// TIA Portal project "PLCwirelessCtrl" (V17)

(* hardware
DEVICE "ET 200SP-Station_1"  ET 200SP-Station
   slot 0: "Baugruppenträger_0"  Rack  6ES5 710-8MAx1
   slot 1: "PLC_1"  CPU 1510SP-1 PN  6ES7 510-1DJ01-0AB0  V2.5
      slot 32768: "PROFINET-Schnittstelle_1"  X1
         slot 32771: "Port_3"  X1 P3
   slot 2: "Servermodul_1"  Server module  6ES7 193-6PA00-0AA0  V1.1
      slot 1: "Servermodul_1"  Server module
   slot 127: "BA 2xRJ45"  BA 2xRJ45  6ES7 193-6AR00-0AA0  V0.0
      slot 32769: "Port_1"  X1 P1  6ES7 193-6AR00-0AA0
      slot 32770: "Port_2"  X1 P2  6ES7 193-6AR00-0AA0
*)

// ===== PLC "PLC_1"  CPU 1510SP-1 PN =====

VAR_GLOBAL   // PLC tag table "Standard-Variablentabelle"
   "Tag_1" AT %M10.1 : Bool;
END_VAR

TYPE "stateBool"
   STRUCT
      "name" : String;
      value : Bool := false;
      alarm : Bool;
      visible : Bool;
      "type" : String := 'bool';
      si : String;
   END_STRUCT;
END_TYPE

TYPE "stateInt"
   STRUCT
      "name" : String;
      value : Int := 52;
      alarm : Bool;
      visible : Bool;
      "type" : String;
      si : String;
   END_STRUCT;
END_TYPE

TYPE "stateReal"
   STRUCT
      "name" : String;
      value : Real := 456.43;
      alarm : Bool;
      visible : Bool;
      "type" : String;
      si : String := '[mbar]';
   END_STRUCT;
END_TYPE

TYPE "paraInt"
   STRUCT
      "name" : String;
      value : Int := 0;
      input : Int;
      locked : Bool := false;
      min : Int := 0;
      max : Int := 9999;
      visible : Bool := true;
      newVal : Bool;
      "type" : String := 'int';
      add : String;
      si : String;
      new : Bool;
   END_STRUCT;
END_TYPE

TYPE "paraBool"
   STRUCT
      "name" : String;
      value : Bool := 0;
      input : Bool;
      locked : Bool := false;
      min : Int := 0;
      max : Int := 1;
      visible : Bool := true;
      newVal : Bool;
      "type" : String := 'bool';
      add : String;
      si : String;
      new : Bool;
   END_STRUCT;
END_TYPE

TYPE "paraReal"
   STRUCT
      "name" : String;
      value : Real := 0.0;
      input : Real;
      locked : Bool := false;
      min : Real := 0.0;
      max : Real := 9999.99;
      visible : Bool := true;
      newVal : Bool;
      "type" : String := 'real';
      add : String;
      si : String;
      new : Bool;
   END_STRUCT;
END_TYPE

TYPE "function"
   STRUCT
      "name" : String;
      active : Bool;
      locked : Bool;
      visible : Bool;
      fault : Bool;
      button : Bool;
      add : Bool;
   END_STRUCT;
END_TYPE

DATA_BLOCK "handleWebserverDat_DB"   // DB1
{ S7_Optimized_Access := 'TRUE' }
VERSION : 0.1
// stored: InstanceOfName handleWebserverDat
"handleWebserverDat"
BEGIN
END_DATA_BLOCK

DATA_BLOCK "webserverData"   // DB3
{ S7_Optimized_Access := 'TRUE' }
VERSION : 0.1
   VAR
      fct00 : "function";
      fct01 : "function";
      fct02 : "function";
      fct03 : "function";
      fct04 : "function";
      fct05 : "function";
      fct06 : "function";
      fct07 : "function";
      fct08 : "function";
      fct09 : "function";
      par00 : "paraInt";
      par01 : "paraBool";
      par02 : "paraReal";
      par03 : "paraInt";
      par04 : "paraInt";
      par05 : "paraInt";
      par06 : "paraInt";
      par07 : "paraInt";
      par08 : "paraInt";
      par09 : "paraInt";
      sta01 : "stateBool";
      sta00 : "stateReal";
      sta02 : "stateBool";
      sta03 : "stateBool";
      sta04 : "stateBool";
      sta05 : "stateBool";
      sta06 : "stateBool";
      sta07 : "stateInt";
      sta08 : "stateBool";
      sta09 : "stateBool";
      alr : Array[0..19] of String;
   END_VAR
BEGIN
   par00."name" := 'Setpoint 1';
   par00."type" := 'int';
   sta01.visible := TRUE;
   sta00."name" := 'Pressure Value';
   sta00.visible := TRUE;
   sta02.value := TRUE;
   sta02.visible := TRUE;
   sta02."type" := 'bool';
   sta07."name" := 'Integer Number';
   sta07.value := 523;
   sta07.si := 'Dig';
   sta01.si := 'Seconds';
   sta01."name" := 'Status of Function';
   par00.min := 0;
   par00.max := 100;
   par00.si := 'cycles';
   par01."name" := 'Manual Mode';
   par02."name" := 'Level';
   par02.si := 'm';
   par02.min := 0.0;
   par02.max := 2000.0;
   par02.locked := TRUE;
   par03."name" := 'Locked Parameter';
   par03.min := 60;
   par03.max := 70;
   par03.locked := TRUE;
   par03.si := 'rpm';
   fct00.visible := TRUE;
   fct01.active := TRUE;
   fct02.locked := TRUE;
   fct03.active := TRUE;
   fct03.locked := TRUE;
   fct03.visible := TRUE;
   fct02.visible := TRUE;
   fct01.visible := TRUE;
   fct04.visible := TRUE;
   fct04.fault := TRUE;
   fct00."name" := 'Function 1';
   fct01."name" := 'Function 2';
   fct02."name" := 'Activate Pump';
   fct03."name" := 'Start Purge';
   fct04."name" := 'Function in Error';
   fct05."name" := 'Reset';
   fct06."name" := 'Do Something';
   fct07."name" := 'Function 8';
   fct08."name" := 'Not Visible';
   fct09."name" := 'Function 10';
   fct09.visible := TRUE;
   fct06.visible := TRUE;
   fct07.visible := TRUE;
   fct05.visible := TRUE;
   sta01."type" := 'bool';
   sta06."name" := 'Distance';
   sta06."type" := 'bool';
   sta06.si := 'm';
   sta00.si := '(mbar)';
   fct00.active := FALSE;
   fct00.locked := FALSE;
   fct00.fault := FALSE;
   fct00.button := FALSE;
   fct00.add := FALSE;
   fct01.locked := FALSE;
   fct01.fault := FALSE;
   fct01.button := FALSE;
   fct01.add := FALSE;
   fct02.active := FALSE;
   fct02.fault := FALSE;
   fct02.button := FALSE;
   fct02.add := FALSE;
   fct03.fault := FALSE;
   fct03.button := FALSE;
   fct03.add := FALSE;
   fct04.active := FALSE;
   fct04.locked := FALSE;
   fct04.button := FALSE;
   fct04.add := FALSE;
   fct05.active := FALSE;
   fct05.locked := FALSE;
   fct05.fault := FALSE;
   fct05.button := FALSE;
   fct05.add := FALSE;
   fct06.active := FALSE;
   fct06.locked := FALSE;
   fct06.fault := FALSE;
   fct06.button := FALSE;
   fct06.add := FALSE;
   fct07.active := FALSE;
   fct07.locked := FALSE;
   fct07.fault := FALSE;
   fct07.button := FALSE;
   fct07.add := FALSE;
   fct08.active := FALSE;
   fct08.locked := FALSE;
   fct08.visible := FALSE;
   fct08.fault := FALSE;
   fct08.button := FALSE;
   fct08.add := FALSE;
   fct09.active := FALSE;
   fct09.locked := FALSE;
   fct09.fault := FALSE;
   fct09.button := FALSE;
   fct09.add := FALSE;
   par00.value := 0;
   par00.input := 0;
   par00.locked := FALSE;
   par00.visible := TRUE;
   par00.newVal := FALSE;
   par00.add := '';
   par00.new := FALSE;
   par01.value := FALSE;
   par01.input := FALSE;
   par01.locked := FALSE;
   par01.min := 0;
   par01.max := 1;
   par01.visible := TRUE;
   par01.newVal := FALSE;
   par01."type" := 'bool';
   par01.add := '';
   par01.si := '';
   par01.new := FALSE;
   par02.value := 0.0;
   par02.input := 0.0;
   par02.visible := TRUE;
   par02.newVal := FALSE;
   par02."type" := 'real';
   par02.add := '';
   par02.new := FALSE;
   par03.value := 0;
   par03.input := 0;
   par03.visible := TRUE;
   par03.newVal := FALSE;
   par03."type" := 'int';
   par03.add := '';
   par03.new := FALSE;
   par04."name" := '';
   par04.value := 0;
   par04.input := 0;
   par04.locked := FALSE;
   par04.min := 0;
   par04.max := 9999;
   par04.visible := FALSE;
   par04.newVal := FALSE;
   par04."type" := 'int';
   par04.add := '';
   par04.si := '';
   par04.new := FALSE;
   par05."name" := '';
   par05.value := 0;
   par05.input := 0;
   par05.locked := FALSE;
   par05.min := 0;
   par05.max := 9999;
   par05.visible := FALSE;
   par05.newVal := FALSE;
   par05."type" := 'int';
   par05.add := '';
   par05.si := '';
   par05.new := FALSE;
   par06."name" := '';
   par06.value := 0;
   par06.input := 0;
   par06.locked := FALSE;
   par06.min := 0;
   par06.max := 9999;
   par06.visible := FALSE;
   par06.newVal := FALSE;
   par06."type" := 'int';
   par06.add := '';
   par06.si := '';
   par06.new := FALSE;
   par07."name" := '';
   par07.value := 0;
   par07.input := 0;
   par07.locked := FALSE;
   par07.min := 0;
   par07.max := 9999;
   par07.visible := FALSE;
   par07.newVal := FALSE;
   par07."type" := 'int';
   par07.add := '';
   par07.si := '';
   par07.new := FALSE;
   par08."name" := '';
   par08.value := 0;
   par08.input := 0;
   par08.locked := FALSE;
   par08.min := 0;
   par08.max := 9999;
   par08.visible := FALSE;
   par08.newVal := FALSE;
   par08."type" := 'int';
   par08.add := '';
   par08.si := '';
   par08.new := FALSE;
   par09."name" := '';
   par09.value := 0;
   par09.input := 0;
   par09.locked := FALSE;
   par09.min := 0;
   par09.max := 9999;
   par09.visible := FALSE;
   par09.newVal := FALSE;
   par09."type" := 'int';
   par09.add := '';
   par09.si := '';
   par09.new := FALSE;
   sta01.value := TRUE;
   sta01.alarm := FALSE;
   sta00.value := 456.43;
   sta00.alarm := FALSE;
   sta00."type" := '';
   sta02."name" := 'Status Pump';
   sta02.alarm := FALSE;
   sta02.si := '';
   sta03."name" := '';
   sta03.value := FALSE;
   sta03.alarm := FALSE;
   sta03.visible := FALSE;
   sta03."type" := 'bool';
   sta03.si := '';
   sta04."name" := '';
   sta04.value := FALSE;
   sta04.alarm := FALSE;
   sta04.visible := FALSE;
   sta04."type" := 'bool';
   sta04.si := '';
   sta05."name" := '';
   sta05.value := FALSE;
   sta05.alarm := FALSE;
   sta05.visible := FALSE;
   sta05."type" := 'bool';
   sta05.si := '';
   sta06.value := FALSE;
   sta06.alarm := FALSE;
   sta06.visible := FALSE;
   sta07.alarm := FALSE;
   sta07.visible := TRUE;
   sta07."type" := '';
   sta08."name" := '';
   sta08.value := FALSE;
   sta08.alarm := FALSE;
   sta08.visible := FALSE;
   sta08."type" := 'bool';
   sta08.si := '';
   sta09."name" := '';
   sta09.value := FALSE;
   sta09.alarm := FALSE;
   sta09.visible := FALSE;
   sta09."type" := 'bool';
   sta09.si := '';
END_DATA_BLOCK

// folder: System blocks/Program resources

DATA_BLOCK "PLC_Control"   // DB332
{ S7_Optimized_Access := 'TRUE' }
VERSION : 0.1
   VAR
      test : Bool;
      test2 : Real;
   END_VAR
BEGIN
END_DATA_BLOCK

// folder: (top level)

FUNCTION_BLOCK "handleWebserverDat"   // FB1, SCL
{ S7_Optimized_Access := 'TRUE' }
VERSION : 0.1
   VAR
      tofPar00 : TOF_TIME;
      tofPar01 : TOF_TIME;
      tofPar02 : TOF_TIME;
      tofPar03 : TOF_TIME;
      tofPar04 : TOF_TIME;
      tofPar05 : TOF_TIME;
      tofPar06 : TOF_TIME;
      tofPar07 : TOF_TIME;
      tofPar08 : TOF_TIME;
      tofPar09 : TOF_TIME;
   END_VAR
BEGIN

   IF "webserverData".par00.new THEN
       "webserverData".par00.value := "webserverData".par00.input;
       "webserverData".par00.newVal := TRUE;
   END_IF;
   #tofPar00(PT := T#1100ms,
             IN := "webserverData".par00.new);
   IF NOT #tofPar00.Q THEN
       "webserverData".par00.newVal := FALSE;
       "webserverData".par00.new := FALSE;
   END_IF;

   IF "webserverData".par01.new THEN
       "webserverData".par01.value := "webserverData".par01.input;
       "webserverData".par01.newVal := TRUE;
   END_IF;
   #tofPar01(PT := T#1100ms,
             IN := "webserverData".par01.new);
   IF NOT #tofPar01.Q THEN
       "webserverData".par01.newVal := FALSE;
       "webserverData".par01.new := FALSE;
   END_IF;

   IF "webserverData".par02.new THEN
       "webserverData".par02.value := "webserverData".par02.input;
       "webserverData".par02.newVal := TRUE;
   END_IF;
   #tofPar02(PT := T#1100ms,
             IN := "webserverData".par02.new);
   IF NOT #tofPar02.Q THEN
       "webserverData".par02.newVal := FALSE;
       "webserverData".par02.new := FALSE;
   END_IF;

   IF "webserverData".par03.new THEN
       "webserverData".par03.value := "webserverData".par03.input;
       "webserverData".par03.newVal := TRUE;
   END_IF;
   #tofPar03(PT := T#1100ms,
             IN := "webserverData".par03.new);
   IF NOT #tofPar03.Q THEN
       "webserverData".par03.newVal := FALSE;
       "webserverData".par03.new := FALSE;
   END_IF;

   IF "webserverData".par04.new THEN
       "webserverData".par04.value := "webserverData".par04.input;
       "webserverData".par04.newVal := TRUE;
   END_IF;
   #tofPar04(PT := T#1100ms,
             IN := "webserverData".par04.new);
   IF NOT #tofPar04.Q THEN
       "webserverData".par04.newVal := FALSE;
       "webserverData".par04.new := FALSE;
   END_IF;

   IF "webserverData".par05.new THEN
       "webserverData".par05.value := "webserverData".par05.input;
       "webserverData".par05.newVal := TRUE;
   END_IF;
   #tofPar05(PT := T#1100ms,
             IN := "webserverData".par05.new);
   IF NOT #tofPar05.Q THEN
       "webserverData".par05.newVal := FALSE;
       "webserverData".par05.new := FALSE;
   END_IF;

   IF "webserverData".par06.new THEN
       "webserverData".par06.value := "webserverData".par06.input;
       "webserverData".par06.newVal := TRUE;
   END_IF;
   #tofPar06(PT := T#1100ms,
             IN := "webserverData".par06.new);
   IF NOT #tofPar06.Q THEN
       "webserverData".par06.newVal := FALSE;
       "webserverData".par06.new := FALSE;
   END_IF;

   IF "webserverData".par07.new THEN
       "webserverData".par07.value := "webserverData".par07.input;
       "webserverData".par07.newVal := TRUE;
   END_IF;
   #tofPar07(PT := T#1100ms,
             IN := "webserverData".par07.new);
   IF NOT #tofPar07.Q THEN
       "webserverData".par07.newVal := FALSE;
       "webserverData".par07.new := FALSE;
   END_IF;

   IF "webserverData".par08.new THEN
       "webserverData".par08.value := "webserverData".par08.input;
       "webserverData".par08.newVal := TRUE;
   END_IF;
   #tofPar08(PT := T#1100ms,
             IN := "webserverData".par08.new);
   IF NOT #tofPar08.Q THEN
       "webserverData".par08.newVal := FALSE;
       "webserverData".par08.new := FALSE;
   END_IF;

   IF "webserverData".par09.new THEN
       "webserverData".par09.value := "webserverData".par09.input;
       "webserverData".par09.newVal := TRUE;
   END_IF;
   #tofPar09(PT := T#1100ms,
             IN := "webserverData".par09.new);
   IF NOT #tofPar09.Q THEN
       "webserverData".par09.newVal := FALSE;
       "webserverData".par09.new := FALSE;
   END_IF;

   IF "webserverData".fct00.button THEN
       "webserverData".fct00.active := NOT "webserverData".fct00.active;
       "webserverData".fct00.button := FALSE;
   END_IF;

   IF "webserverData".fct01.button THEN
       "webserverData".fct01.active := NOT "webserverData".fct01.active;
       "webserverData".fct01.button := FALSE;
   END_IF;

   IF "webserverData".fct02.button THEN
       "webserverData".fct02.active := NOT "webserverData".fct02.active;
       "webserverData".fct02.button := FALSE;
   END_IF;

   IF "webserverData".fct03.button THEN
       "webserverData".fct03.active := NOT "webserverData".fct03.active;
       "webserverData".fct03.button := FALSE;
   END_IF;

   IF "webserverData".fct04.button THEN
       "webserverData".fct04.active := NOT "webserverData".fct04.active;
       "webserverData".fct04.button := FALSE;
   END_IF;

   IF "webserverData".fct05.button THEN
       "webserverData".fct05.active := NOT "webserverData".fct05.active;
       "webserverData".fct05.button := FALSE;
   END_IF;

   IF "webserverData".fct06.button THEN
       "webserverData".fct06.active := NOT "webserverData".fct06.active;
       "webserverData".fct06.button := FALSE;
   END_IF;

   IF "webserverData".fct07.button THEN
       "webserverData".fct07.active := NOT "webserverData".fct07.active;
       "webserverData".fct07.button := FALSE;
   END_IF;

   IF "webserverData".fct08.button THEN
       "webserverData".fct08.active := NOT "webserverData".fct08.active;
       "webserverData".fct08.button := FALSE;
   END_IF;

   IF "webserverData".fct09.button THEN
       "webserverData".fct09.active := NOT "webserverData".fct09.active;
       "webserverData".fct09.button := FALSE;
   END_IF;
END_FUNCTION_BLOCK

ORGANIZATION_BLOCK "Main"   // OB1, LAD, ProgramCycle
TITLE = "Main Program Sweep (Cycle)"
{ S7_Optimized_Access := 'TRUE' }
VERSION : 0.1
   VAR_INPUT
      Initial_Call : Bool;   // Initial call of this OB
      Remanence : Bool;   // =True, if remanent data are available
   END_VAR
   VAR_TEMP
      temp : Int;
   END_VAR
BEGIN

REGION Network 1
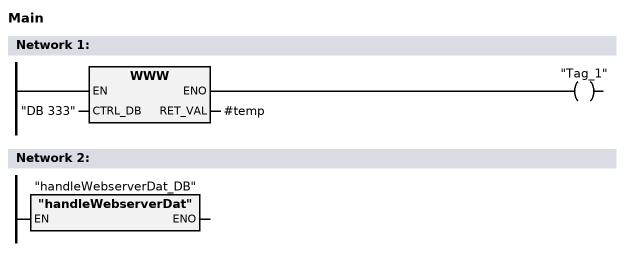
   // ENO of a box is taken as its EN; it also drops when the box reports an error
   #temp := WWW(CTRL_DB := "DB 333");
   "Tag_1" := TRUE;
END_REGION

REGION Network 2
   RUNG wire#powerrail
      "handleWebserverDat_DB"()
   END_RUNG
   // the same network as SCL:
   "handleWebserverDat_DB"();   // "handleWebserverDat"
END_REGION
END_ORGANIZATION_BLOCK